(* CoDeSys 2.3.9.37 project: Cap10_2.pro *)
(* Libraries: Standard.lib 4.10.05 12:14:46 *)

(* Global variable list: Global_Variables *)
VAR_GLOBAL
    (*Entradas *)
    Abre : BOOL;  (* Pulsador que se usará para abrir la válvula *)
    Cierra : BOOL;  (* Pulsadir para cerrar la válvula *)
    FCA : BOOL; (* Fin de carrera apertura *)
    FCC : BOOL;  (* Fin de carrera cierre *)
    (* Salidas*)
    Bobina : BOOL;  (* Bovina de la válvula 2/2 *)
    ErrorValvula : BOOL;  (* Luz de aviso error *)
END_VAR

(* POU PLC_PRG, FBD *)
PROGRAM PLC_PRG
VAR
END_VAR
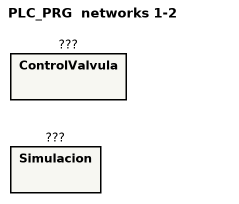
_FBD_ (* Function Block Diagram *)
NETWORK 1
	???:ControlValvula()
NETWORK 2
	???:Simulacion()
_END_FBD_
END_PROGRAM

(* POU ControlValvula, FBD *)
PROGRAM ControlValvula
VAR
END_VAR
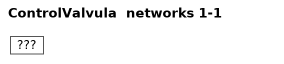
_FBD_ (* Function Block Diagram *)
NETWORK 1
	???
_END_FBD_
(* the same logic as Structured Text *)
(* Network 1 *)
END_PROGRAM

(* POU Simulacion, ST *)
PROGRAM Simulacion
VAR
   PosVal : INT;
   FALLO:BOOL;
END_VAR
IF Bobina AND (PosVal>-50) AND (NOT FALLO)  THEN
   PosVal:=PosVal-1;
END_IF

IF (NOT Bobina) AND PosVal<=0 AND (NOT FALLO) THEN
   PosVal:=PosVal+1;
END_IF

 FCC:= (PosVal>=0);
FCA:=(PosVal<=-50);
END_PROGRAM

(* Visualisation Valvula
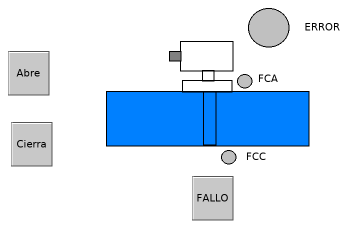
button at (68,56)-(109,100): text "Abre"; taps Abre
button at (71,127)-(112,171): text "Cierra"; taps Cierra
rectangle at (263,96)-(276,150): bottom Simulacion.PosVal
rounded rectangle at (229,56)-(241,66): alarm colour if Bobina
ellipse at (281,155)-(296,169): alarm colour if FCC
ellipse at (297,79)-(312,93): alarm colour if FCA
rectangle at (300,152)-(332,171): text "FCC"
rectangle at (312,74)-(344,93): text "FCA"
button at (252,181)-(293,225): text "FALLO"; toggles Simulacion.FALLO
ellipse at (308,13)-(349,52): alarm colour if ErrorValvula
rectangle at (355,18)-(410,46): text "ERROR"
4 more shapes without text or variables
*)
